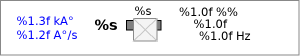
VISUALIZATION VISU_XTAL_6  // 300x56
VAR_IN_OUT
	m_Input_XTAL : BLOCK_XTAL6;
END_VAR

VAR_INPUT
	m_Input_NumFrame_Manu:	USINT;		(*numéro de frame à afficher dans le synoptique MANUEL*)
END_VAR
    Rectangle (0,0 300x56)
        OnMouseClick: execute { .VISU_INDEX_MANU := m_Input_NumFrame_Manu; }
        OnMouseClick: change screen: SYN_MANUEL
    Rectangle (1,14 85x14), "%1.3f kA°", text variable: m_Input_XTAL.STATE_THICKNESS
    Rectangle (125,3 36x16), "%s", text variable: m_Input_XTAL.MNEMO
    Rectangle (126,20 35x10)
    RoundedRectangle (136,28 17x7)
    Rectangle (164,5 86x14), "%1.0f %%", text variable: m_Input_XTAL.STATE_ACTUAL_CRYS_LIFE
    Rectangle (163,29 120x14), "%1.0f Hz", text variable: m_Input_XTAL.STATE_ACTUAL_CRYS_FREQ
    Rectangle (164,17 89x14), "%1.0f", text variable: m_Input_XTAL.STATE_ACTUAL_CRYS_ACTIVITY
    Rectangle (3,28 85x14), "%1.2f A°/s", text variable: m_Input_XTAL.STATE_RATE
    Image (133,18 24x23), invisible if: NOT m_Input_XTAL.STATE_NOK, image: MesImages.warning
    Rectangle (86,16 40x18), "%s", text variable: m_Input_XTAL.STATE_POSITION
END_VISUALIZATION

(* stored: Version 1.1.0.1, ProductVersion 3.1.4024.11
   Visu VISU_XTAL_6: Id {a8c123e3-4f5c-4072-9213-f77f6b96e158} *)
